// TIA Portal V20 export
ORGANIZATION_BLOCK "Cyclic interrupt_1"   // OB31, LAD, CyclicInterrupt
{ S7_Optimized_Access := 'TRUE' }
// stored: SetENOAutomatically false
   VAR_INPUT
      Initial_Call : Bool;   // Initial call of this OB
      Event_Count : Int;   // Events discarded
   END_VAR
BEGIN

REGION Network 1 (SCL)
   // "DB_MC2".Status := -1;
END_REGION
END_ORGANIZATION_BLOCK
